{attribute addProperty BoxType "EL6201-0000-0017"}
{attribute addProperty Id "Slave_8A_DI0BIT10.12557Slave_8A_DI1BIT10.12558Slave_8A_DI2BIT10.12559Slave_8A_DI3BIT10.12560Slave_8B_DI0BIT10.12561Slave_8B_DI1BIT10.12562Slave_8B_DI2BIT10.12563Slave_8B_DI3BIT10.12564"}
{attribute addProperty CRC "2693962661"}
{attribute addProperty SizeInBites "8"}
{attribute addProperty SizeInBytes "1"}
TYPE Slave_8_Inputs_A0929BA5 :
STRUCT
	{attribute addProperty Name "Slave_8A_DI0"}
	Slave_8A_DI0 : BIT;
	{attribute addProperty Name "Slave_8A_DI1"}
	Slave_8A_DI1 : BIT;
	{attribute addProperty Name "Slave_8A_DI2"}
	Slave_8A_DI2 : BIT;
	{attribute addProperty Name "Slave_8A_DI3"}
	Slave_8A_DI3 : BIT;
	{attribute addProperty Name "Slave_8B_DI0"}
	Slave_8B_DI0 : BIT;
	{attribute addProperty Name "Slave_8B_DI1"}
	Slave_8B_DI1 : BIT;
	{attribute addProperty Name "Slave_8B_DI2"}
	Slave_8B_DI2 : BIT;
	{attribute addProperty Name "Slave_8B_DI3"}
	Slave_8B_DI3 : BIT;
END_STRUCT
END_TYPE

(* stored: Version 1.2.0.0, ProductVersion 3.1.4024.9
   DUT Slave_8_Inputs_A0929BA5: Id {ff04e7e5-539e-40cb-b0a6-782bc48c25c2} *)
